FUNCTION_BLOCK FB_RobotArmPickAndPlace EXTENDS FB_RobotArm
VAR
	
END_VAR

SUPER^();

METHOD PUBLIC M_PickUpFromPlace : BOOL
VAR_INPUT
	PLACE_NUM 	: INT;
END_VAR

VAR_INST
	Step		: INT := 0;
END_VAR
CASE PLACE_NUM OF
	E_BoxPlaceDirection.PLACE1_LEFT: //IF  place1 NOT empty
		Step := E_PickPlaceStep.MOVE_HAND;
		CASE Step OF
			E_PickPlaceStep.DO_NOTHING:
				// do nothing
			E_PickPlaceStep.MOVE_HAND:
				FOR Index := 1 TO BaseConfiguration.NUMBER_OF_JOINTS BY 1 DO
					M_TurnJoint( TurnDirection := E_RobotArmJointDirection.LEFT, Joint := Index);
					
					IF NOT InputsDecoupled.JOINT_LEFT_SIGNAL[Index] THEN
						Index := Index - 1;
					END_IF
				END_FOR
				
				Step := E_PickPlaceStep.CHECK_GRIP;
			
			E_PickPlaceStep.CHECK_GRIP:
				IF InputsDecoupled.GRIP_CLOSED THEN
					Outputs.GRIP_CLOSE := FALSE;
				ELSE
					Step := E_PickPlaceStep.USE_GRIP;
				END_IF
				
			E_PickPlaceStep.USE_GRIP:
				IF NOT InputsDecoupled.GRIP_CLOSED THEN
					Outputs.GRIP_CLOSE := TRUE;
					Step := E_PickPlaceStep.DO_NOTHING;
					PLACE_NUM := E_BoxPlaceDirection.UNDEFINED;
				END_IF
				
		END_CASE
	
	E_BoxPlaceDirection.PLACE2_RIGHT: // //IF  place2 empty
		
	
END_CASE
END_METHOD

METHOD PUBLIC M_PlaceTo : BOOL
VAR_INPUT
	PLACE_NUM : INT;
END_VAR
END_METHOD

END_FUNCTION_BLOCK

(* stored: Version 1.1.0.1, ProductVersion 3.1.4024.9
   POU FB_RobotArmPickAndPlace: Id {842cc1cd-ba85-4d04-97c1-8be629b74f41}, SpecialFunc None
   Method M_PickUpFromPlace: Id {0d7a498c-12eb-4758-998c-0b68373ba906}
   Method M_PlaceTo: Id {ae78284d-df5e-4770-a799-68f8df794d6d} *)
